TYPE Result_Status :
STRUCT
	Decoding			  : BOOL;
	Decode_Complete 	  : BOOL;
	Result_Buffer_overrun : BOOL;
	Result_Available	  : BOOL;
	Set_When_fault_Occur  : BOOL;
END_STRUCT
END_TYPE

(* stored: Version 1.1.0.1, ProductVersion 3.1.4024.11
   DUT Result_Status: Id {a7769bb6-274b-46ed-8a76-e23378c6c02d} *)
